PROGRAM MAIN
VAR
	Stopwatch1 : FB_StopWatch_Level;
END_VAR

Stopwatch1(bSTART:= , bRESET:= , Elapsed_Time=> );

END_PROGRAM

(* stored: Version 1.1.0.1, ProductVersion 3.1.4024.5
   POU MAIN: Id {a0f2ab23-8e12-45a0-b18b-744a7b3e2756}, SpecialFunc None *)
